// TIA Portal V19 export
VAR_GLOBAL   // PLC tag table "Dispenser_Tags"
   Power_ON AT %M1.0 : Bool;   // Power on Command
   Power_OFF AT %M1.1 : Bool;   // Power off Command
   Power_Active AT %M1.2 : Bool;   // Power is Active
   Start AT %M1.3 : Bool;   // Start Command
   Motor AT %M1.5 : Bool;   // Motor Status
   Gate1 AT %M1.6 : Bool;   // Light Gate Sensor 1
   Gate2 AT %M1.7 : Bool;   // Light Gate Sensor 2
   Gate3 AT %M2.0 : Bool;   // Light Gate Sensor 3
   Gate4 AT %M2.1 : Bool;   // Light Gate Sensor 4
   Gate5 AT %M2.2 : Bool;   // Light Gate Sensor 5
   Dropper_A AT %M2.3 : Bool;   // Dispenser Dropper 1
   Dropper_B AT %M2.4 : Bool;   // Dispenser Dropper 2
   Dropper_C AT %M2.5 : Bool;   // Dispenser Dropper 3
   Stop AT %M1.4 : Bool;   // Stop Command
   SW_A AT %M2.6 : Bool;   // Switch A
   SW_B AT %M2.7 : Bool;   // Switch B
   SW_C AT %M3.0 : Bool;   // Switch C
   Process_Started AT %M3.1 : Bool;   // Dispenser Process Running
   StopDispenser AT %M3.2 : Bool;   // E-Stop for Dispenser
END_VAR
